INTERFACE I_MotionAxisPower


METHOD GetMode : E_MotionAxisPowerMode
END_METHOD


METHOD PowerOff
END_METHOD


METHOD PowerOn
END_METHOD

END_INTERFACE

(* stored: Version 1.1.0.1
   Itf I_MotionAxisPower: Id {574f915f-b873-4905-bd65-b4e43afdffdc}
   Method GetMode: Id {d3591742-e354-4fe0-bf0f-8ade5f478837}
   Method PowerOff: Id {0667cdd9-efe4-424e-9f73-3f99ff97713f}
   Method PowerOn: Id {a1fe0419-6a20-4fae-8aa7-85ee393666ff} *)
